# EPICS autosave request: autosave/galil_user_array.req
$(P)UARRAYNAME$(ADDR)_SP
